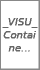
VISUALIZATION VISU_CTFlow  // 40x70
VAR_IN_OUT
	m_Inst  : FB_CTManagerView;
END_VAR
    Frame (0,0 40x70)
        shows _VISU_ContainerView(m_Inst := m_Inst.aCTV[1])
        p3560616238: m_Inst.aCTV[1]._posX
        p2738717112: m_Inst.aCTV[1]._posY
    Frame (0,0 40x70)
        shows _VISU_ContainerView(m_Inst := m_Inst.aCTV[2])
        p3560616238: m_Inst.aCTV[2]._posX
        p2738717112: m_Inst.aCTV[2]._posY
    Frame (0,0 40x70)
        shows _VISU_ContainerView(m_Inst := m_Inst.aCTV[3])
        p3560616238: m_Inst.aCTV[3]._posX
        p2738717112: m_Inst.aCTV[3]._posY
    Frame (0,0 40x70)
        shows _VISU_ContainerView(m_Inst := m_Inst.aCTV[4])
        p3560616238: m_Inst.aCTV[4]._posX
        p2738717112: m_Inst.aCTV[4]._posY
    Frame (0,0 40x70)
        shows _VISU_ContainerView(m_Inst := m_Inst.aCTV[5])
        p3560616238: m_Inst.aCTV[5]._posX
        p2738717112: m_Inst.aCTV[5]._posY
    Frame (0,0 40x70)
        shows _VISU_ContainerView(m_Inst := m_Inst.aCTV[6])
        p3560616238: m_Inst.aCTV[6]._posX
        p2738717112: m_Inst.aCTV[6]._posY
    Frame (0,0 40x70)
        shows _VISU_ContainerView(m_Inst := m_Inst.aCTV[7])
        p3560616238: m_Inst.aCTV[7]._posX
        p2738717112: m_Inst.aCTV[7]._posY
    Frame (0,0 40x70)
        shows _VISU_ContainerView(m_Inst := m_Inst.aCTV[8])
        p3560616238: m_Inst.aCTV[8]._posX
        p2738717112: m_Inst.aCTV[8]._posY
    Frame (0,0 40x70)
        shows _VISU_ContainerView(m_Inst := m_Inst.aCTV[9])
        p3560616238: m_Inst.aCTV[9]._posX
        p2738717112: m_Inst.aCTV[9]._posY
    Frame (0,0 40x70)
        shows _VISU_ContainerView(m_Inst := m_Inst.aCTV[10])
        p3560616238: m_Inst.aCTV[10]._posX
        p2738717112: m_Inst.aCTV[10]._posY
    Frame (0,0 40x70)
        shows _VISU_ContainerView(m_Inst := m_Inst.aCTV[11])
        p3560616238: m_Inst.aCTV[11]._posX
        p2738717112: m_Inst.aCTV[11]._posY
    Frame (0,0 40x70)
        shows _VISU_ContainerView(m_Inst := m_Inst.aCTV[12])
        p3560616238: m_Inst.aCTV[12]._posX
        p2738717112: m_Inst.aCTV[12]._posY
    Frame (0,0 40x70)
        shows _VISU_ContainerView(m_Inst := m_Inst.aCTV[13])
        p3560616238: m_Inst.aCTV[13]._posX
        p2738717112: m_Inst.aCTV[13]._posY
    Frame (0,0 40x70)
        shows _VISU_ContainerView(m_Inst := m_Inst.aCTV[14])
        p3560616238: m_Inst.aCTV[14]._posX
        p2738717112: m_Inst.aCTV[14]._posY
    Frame (0,0 40x70)
        shows _VISU_ContainerView(m_Inst := m_Inst.aCTV[15])
        p3560616238: m_Inst.aCTV[15]._posX
        p2738717112: m_Inst.aCTV[15]._posY
    Frame (0,0 40x70)
        shows _VISU_ContainerView(m_Inst := m_Inst.aCTV[16])
        p3560616238: m_Inst.aCTV[16]._posX
        p2738717112: m_Inst.aCTV[16]._posY
    Frame (0,0 40x70)
        shows _VISU_ContainerView(m_Inst := m_Inst.aCTV[17])
        p3560616238: m_Inst.aCTV[17]._posX
        p2738717112: m_Inst.aCTV[17]._posY
    Frame (0,0 40x70)
        shows _VISU_ContainerView(m_Inst := m_Inst.aCTV[18])
        p3560616238: m_Inst.aCTV[18]._posX
        p2738717112: m_Inst.aCTV[18]._posY
    Frame (0,0 40x70)
        shows _VISU_ContainerView(m_Inst := m_Inst.aCTV[19])
        p3560616238: m_Inst.aCTV[19]._posX
        p2738717112: m_Inst.aCTV[19]._posY
    Frame (0,0 40x70)
        shows _VISU_ContainerView(m_Inst := m_Inst.aCTV[21])
        p3560616238: m_Inst.aCTV[21]._posX
        p2738717112: m_Inst.aCTV[21]._posY
    Frame (0,0 40x70)
        shows _VISU_ContainerView(m_Inst := m_Inst.aCTV[22])
        p3560616238: m_Inst.aCTV[22]._posX
        p2738717112: m_Inst.aCTV[22]._posY
    Frame (0,0 40x70)
        shows _VISU_ContainerView(m_Inst := m_Inst.aCTV[23])
        p3560616238: m_Inst.aCTV[23]._posX
        p2738717112: m_Inst.aCTV[23]._posY
    Frame (0,0 40x70)
        shows _VISU_ContainerView(m_Inst := m_Inst.aCTV[24])
        p3560616238: m_Inst.aCTV[24]._posX
        p2738717112: m_Inst.aCTV[24]._posY
    Frame (0,0 40x70)
        shows _VISU_ContainerView(m_Inst := m_Inst.aCTV[25])
        p3560616238: m_Inst.aCTV[25]._posX
        p2738717112: m_Inst.aCTV[25]._posY
    Frame (0,0 40x70)
        shows _VISU_ContainerView(m_Inst := m_Inst.aCTV[26])
        p3560616238: m_Inst.aCTV[26]._posX
        p2738717112: m_Inst.aCTV[26]._posY
    Frame (0,0 40x70)
        shows _VISU_ContainerView(m_Inst := m_Inst.aCTV[27])
        p3560616238: m_Inst.aCTV[27]._posX
        p2738717112: m_Inst.aCTV[27]._posY
    Frame (0,0 40x70)
        shows _VISU_ContainerView(m_Inst := m_Inst.aCTV[28])
        p3560616238: m_Inst.aCTV[28]._posX
        p2738717112: m_Inst.aCTV[28]._posY
    Frame (0,0 40x70)
        shows _VISU_ContainerView(m_Inst := m_Inst.aCTV[29])
        p3560616238: m_Inst.aCTV[29]._posX
        p2738717112: m_Inst.aCTV[29]._posY
    Frame (0,0 40x70)
        shows _VISU_ContainerView(m_Inst := m_Inst.aCTV[30])
        p3560616238: m_Inst.aCTV[30]._posX
        p2738717112: m_Inst.aCTV[30]._posY
    Frame (0,0 40x70)
        shows _VISU_ContainerView(m_Inst := m_Inst.aCTV[31])
        p3560616238: m_Inst.aCTV[31]._posX
        p2738717112: m_Inst.aCTV[31]._posY
    Frame (0,0 40x70)
        shows _VISU_ContainerView(m_Inst := m_Inst.aCTV[32])
        p3560616238: m_Inst.aCTV[32]._posX
        p2738717112: m_Inst.aCTV[32]._posY
    Frame (0,0 40x70)
        shows _VISU_ContainerView(m_Inst := m_Inst.aCTV[33])
        p3560616238: m_Inst.aCTV[33]._posX
        p2738717112: m_Inst.aCTV[33]._posY
    Frame (0,0 40x70)
        shows _VISU_ContainerView(m_Inst := m_Inst.aCTV[34])
        p3560616238: m_Inst.aCTV[34]._posX
        p2738717112: m_Inst.aCTV[34]._posY
    Frame (0,0 40x70)
        shows _VISU_ContainerView(m_Inst := m_Inst.aCTV[35])
        p3560616238: m_Inst.aCTV[35]._posX
        p2738717112: m_Inst.aCTV[35]._posY
    Frame (0,0 40x70)
        shows _VISU_ContainerView(m_Inst := m_Inst.aCTV[36])
        p3560616238: m_Inst.aCTV[36]._posX
        p2738717112: m_Inst.aCTV[36]._posY
    Frame (0,0 40x70)
        shows _VISU_ContainerView(m_Inst := m_Inst.aCTV[37])
        p3560616238: m_Inst.aCTV[37]._posX
        p2738717112: m_Inst.aCTV[37]._posY
    Frame (0,0 40x70)
        shows _VISU_ContainerView(m_Inst := m_Inst.aCTV[38])
        p3560616238: m_Inst.aCTV[38]._posX
        p2738717112: m_Inst.aCTV[38]._posY
    Frame (0,0 40x70)
        shows _VISU_ContainerView(m_Inst := m_Inst.aCTV[39])
        p3560616238: m_Inst.aCTV[39]._posX
        p2738717112: m_Inst.aCTV[39]._posY
    Frame (0,0 40x70)
        shows _VISU_ContainerView(m_Inst := m_Inst.aCTV[40])
        p3560616238: m_Inst.aCTV[40]._posX
        p2738717112: m_Inst.aCTV[40]._posY
    Frame (0,0 40x70)
        shows _VISU_ContainerView(m_Inst := m_Inst.aCTV[41])
        p3560616238: m_Inst.aCTV[41]._posX
        p2738717112: m_Inst.aCTV[41]._posY
    Frame (0,0 40x70)
        shows _VISU_ContainerView(m_Inst := m_Inst.aCTV[42])
        p3560616238: m_Inst.aCTV[42]._posX
        p2738717112: m_Inst.aCTV[42]._posY
    Frame (0,0 40x70)
        shows _VISU_ContainerView(m_Inst := m_Inst.aCTV[43])
        p3560616238: m_Inst.aCTV[43]._posX
        p2738717112: m_Inst.aCTV[43]._posY
    Frame (0,0 40x70)
        shows _VISU_ContainerView(m_Inst := m_Inst.aCTV[44])
        p3560616238: m_Inst.aCTV[44]._posX
        p2738717112: m_Inst.aCTV[44]._posY
    Frame (0,0 40x70)
        shows _VISU_ContainerView(m_Inst := m_Inst.aCTV[45])
        p3560616238: m_Inst.aCTV[45]._posX
        p2738717112: m_Inst.aCTV[45]._posY
    Frame (0,0 40x70)
        shows _VISU_ContainerView(m_Inst := m_Inst.aCTV[46])
        p3560616238: m_Inst.aCTV[46]._posX
        p2738717112: m_Inst.aCTV[46]._posY
    Frame (0,0 40x70)
        shows _VISU_ContainerView(m_Inst := m_Inst.aCTV[47])
        p3560616238: m_Inst.aCTV[47]._posX
        p2738717112: m_Inst.aCTV[47]._posY
    Frame (0,0 40x70)
        shows _VISU_ContainerView(m_Inst := m_Inst.aCTV[48])
        p3560616238: m_Inst.aCTV[48]._posX
        p2738717112: m_Inst.aCTV[48]._posY
    Frame (0,0 40x70)
        shows _VISU_ContainerView(m_Inst := m_Inst.aCTV[49])
        p3560616238: m_Inst.aCTV[49]._posX
        p2738717112: m_Inst.aCTV[49]._posY
    Frame (0,0 40x70)
        shows _VISU_ContainerView(m_Inst := m_Inst.aCTV[50])
        p3560616238: m_Inst.aCTV[50]._posX
        p2738717112: m_Inst.aCTV[50]._posY
    Frame (0,0 40x70)
        shows _VISU_ContainerView(m_Inst := m_Inst.aCTV[20])
        p3560616238: m_Inst.aCTV[20]._posX
        p2738717112: m_Inst.aCTV[20]._posY
END_VISUALIZATION

(* stored: Version 1.1.0.1, ProductVersion 3.1.4024.3
   Visu VISU_CTFlow: Id {881136dc-89d7-4d7a-9bec-12bc9ffd62d4} *)
